Staubli VAL3: checkPoint.pgx

public program checkPoint(point x_PointToGo, point x_PointStart, bool& x_bUnreached[], tool x_tTool, bool x_bLinear)
  local joint jpO_frameint
  local string message
  local num i
begin
  // check if the pO_frameint is null???
  if (cycleStatus:bCycle==false and cycleStatus:bSimulation==false) or !x_bLinear
    x_bUnreached=(position(x_PointToGo,world)=={0,0,0,0,0,0})
    //
    if !x_bUnreached
      //
      // look if the pO_frameint that you want to reach is valid
      if x_bLinear
        //
        // use the percentage....
        //
        for i=0.1 to 1 step 0.1
          pCheck.trsf=interpolateL(position(x_PointStart,world),position(x_PointToGo,world),i)
          x_bUnreached=!pointToJoint(x_tTool,herej(),pCheck,jpO_frameint)
          if x_bUnreached
            return
          endIf
        endFor
      else
        // joint move or check only the working area
        x_PointToGo.config={sfree,efree,wfree}
        x_bUnreached=!pointToJoint(x_tTool,herej(),x_PointToGo,jpO_frameint)
      endIf
    endIf
  endIf
end
